(* Logix 5000 project; controller IndiconLLC vendor 1 type 14 code 77 rev 20.14; software revision 20.05 *)
// Indicon Emulation Department CompactLogix
// Development Kit PLC

TASK MainTask (continuous, watchdog 500 ms) : CPU

MODULES
   Controller : vendor 1 type 14 code 77 (CompactLogixL32EController 0, rev 20.14)
      LocalENB : 1769-L32E Ethernet Port (CompactLogixL32Ethernet 1, rev 20.11)
         AS1_ENBT : 1756-ENBT (Ethernet 192.168.112.83, rev 4.7, Output RPI 10 ms)
            AS1 : vendor 1 type 14 code 213 (ICP 2, rev 32.1, $37f21408$ RPI 50 ms)
      Local : CompactBus (CompactVirtualAdapter 3, rev 20.11)
END_MODULES

TYPE Emulation_Carrier_Object :
STRUCT
   Spawned : BOOL;
   XPos : DINT;
   Width : DINT;
   ZeroPoint : DINT;
   EndPoint : DINT;
   RealPosition : REAL;
   RestrictSpawn : BOOL;
   AttachedFront : BOOL;
   AttachedFrontID : DINT;
   AttachedRear : BOOL;
   AttachedRearID : DINT;
   DirectiveFlowFwd : BOOL;
   DirectiveFlowRev : BOOL;
   UpdateCounter : DINT;
END_STRUCT
END_TYPE

TYPE Emulation_Display_Env :
STRUCT
   Height : DINT;
   Width : DINT;
   CarrierObjectWidth : DINT;
   CarrierObjectCountSize : DINT;
   CarrierObjectFORControl : DINT;
   CarrierObjectFORControlEmbed : DINT;
   VFDObjectWidth : DINT;
   VFDObjectCountSize : DINT;
   VFDObjectFORControl : DINT;
END_STRUCT
END_TYPE

TYPE ProdCons_VFD :
STRUCT
   VFD : ProdCons_VFD_PTP_Setup[3];
END_STRUCT
END_TYPE

TYPE ProdCons_VFD_PTP_Setup :
STRUCT
   In : z_VFD_PTP_Emulation_Input;
   Out : z_VFD_PTP_Emulation_Output;
END_STRUCT
END_TYPE

TYPE ProdCons_VFD_Setup :
STRUCT
   In : z_VFD_Emulation_Input;
   Out : z_VFD_Emulation_Output;
END_STRUCT
END_TYPE

TYPE student_DataHandlingVehicleObject :
STRUCT
   Visibility : BOOL;
   YPosition : DINT;
   XPosition : DINT;
   PositionUpdateDwell : TIMER;
   InSpawnZone : BOOL;
   ShiftRegisterData : DINT;
   Color : SINT;
   ONS : DINT;
   DedicatedBank : SINT;
END_STRUCT
END_TYPE

TYPE z_VFD_Emulation :
STRUCT
   OverView : z_VFD_Emulation_Handling;
   MotorOutputs : z_VFD_Emulation_Input;
   MotorInputs : z_VFD_Emulation_Output;
END_STRUCT
END_TYPE

TYPE z_VFD_Emulation_Handling :
STRUCT
   XPosition : DINT;
   YPosition : DINT;
   Width : DINT;
   ZeroPoint : DINT;
   EndPoint : DINT;
   MoveFwd : BOOL;
   MoveRev : BOOL;
   HiSpeed : DINT;
   LoSpeed : DINT;
   HiSpeedEnable : BOOL;
   AccelRamp : DINT;
   DecelRamp : DINT;
   AccelCalc : REAL;
   DecelCalc : REAL;
   CurrentSpeed : REAL;
   SpeedCalc : REAL;
   ForwardLocked : BOOL;
   ReverseLocked : BOOL;
   PositionUpdateDwell : TIMER;
   SpeedDividend : REAL;
   IO : SINT;
   StationType : DINT;
   PXS : z_VFD_Emulation_IO_Handling[6];
   Position : DINT;
END_STRUCT
END_TYPE

TYPE z_VFD_Emulation_Input :
STRUCT
   ReadyToRun : BOOL;
   FaultCode : DINT;
   VelocityFeedback : DINT;
   MotorRunningFwd : BOOL;
   MotorRunningRev : BOOL;
   IO : SINT;
   PositionFeedback : DINT;
END_STRUCT
END_TYPE

TYPE z_VFD_Emulation_IO_Handling :
STRUCT
   Enable : BOOL;
   Position : DINT;
   RequestStuckOnSim : BOOL;
   RequestStuckOffSim : BOOL;
END_STRUCT
END_TYPE

TYPE z_VFD_Emulation_Output :
STRUCT
   RunForward : BOOL;
   RunReverse : BOOL;
   SpeedSetpoint : DINT;
   FaultReset : BOOL;
END_STRUCT
END_TYPE

TYPE z_VFD_PTP_Emulation :
STRUCT
   OverView : z_VFD_Emulation_Handling;
   MotorOutputs : z_VFD_PTP_Emulation_Input;
   MotorInputs : z_VFD_PTP_Emulation_Output;
END_STRUCT
END_TYPE

TYPE z_VFD_PTP_Emulation_Input :
STRUCT
   ReadyToRun : BOOL;
   FaultCode : DINT;
   VelocityFeedback : DINT;
   MotorRunningFwd : BOOL;
   MotorRunningRev : BOOL;
   IO : SINT;
   PositionFeedback : DINT;
END_STRUCT
END_TYPE

TYPE z_VFD_PTP_Emulation_Internal :
STRUCT
   Offset : DINT;
   Position : DINT;
   CaptureOneShot : BOOL;
   ForwardMoveRequired : BOOL;
   ReverseMoveRequired : BOOL;
   HighSpeedEnable : BOOL;
   CreepSpeedEnable : BOOL;
   SpeedLimit : REAL;
   AbsTenPercent : REAL;
   AbsTenPercentNeg : REAL;
   AbsTenPercentEmb : REAL;
   AbsTenPercentEmbNeg : REAL;
   OneShot : DINT;
END_STRUCT
END_TYPE

TYPE z_VFD_PTP_Emulation_Output :
STRUCT
   JogForward : BOOL;
   JogReverse : BOOL;
   SpeedSetpoint : DINT;
   PTPSetpoint : DINT;
   PTP_Move : BOOL;
   Run : BOOL;
   FaultReset : BOOL;
END_STRUCT
END_TYPE

TYPE zFlash :
STRUCT
   Slow : BOOL;
   Norm : BOOL;
   Fast : BOOL;
   Timer : TIMER;
END_STRUCT
END_TYPE

TYPE zTime :
STRUCT
   Year : DINT;
   Month : DINT;
   Day : DINT;
   Hour : DINT;
   Minute : DINT;
   Second : DINT;
   MSecond : DINT;
END_STRUCT
END_TYPE

VAR_GLOBAL   (* controller tags *)
   AS1_ToSupervisor : ProdCons_VFD := (VFD[0].Out.SpeedSetpoint := 500, VFD[0].Out.PTPSetpoint := 7718, VFD[1].Out.SpeedSetpoint := 250, VFD[1].Out.PTPSetpoint := 6082, VFD[2].Out.SpeedSetpoint := 250);
   Flash : zFlash := (Slow := 1, Fast := 1, Timer.PRE := 8388608, Timer.ACC := 3363, Timer.EN := 1, Timer.TT := 1);
   initializeDint : DINT := 100;
   InitializeMessage : MESSAGE;
        MessageParameters(ServiceCode := 16#004d, LocalElement := initializeDint, ...)
   ProducedData : DINT[300] := ([0] := 17);
   ReadWallClock : zTime := (Year := 2019, Month := 5, Day := 15, Hour := 4, Minute := 41, Second := 27, MSecond := 192466);
   Supervisor_ToAS1 : ProdCons_VFD := (VFD[0].In.PositionFeedback := 7718, VFD[1].In.PositionFeedback := 6082, VFD[2].In.PositionFeedback := 4); {produced}
   TempDINT : DINT[1000] := ([0] := 99999999, [1] := 99999999, [2] := 99999999, [3] := 99999999, [4] := 99999999, [5] := 99999999, [6] := 99999999, [7] := 99999999, [8] := 99999999, [9] := 99999999, [10] := 99999999, [11] := 99999999, [12] := 99999999, [13] := 99999999, [14] := 99999999, [15] := 99999999, [16] := 99999999, [17] := 99999999, [18] := 99999999, [19] := 99999999, [20] := 99999999, [21] := 99999999, [22] := 99999999, [23] := 99999999, [24] := 99999999, [25] := 99999999, [26] := 99999999, [27] := 99999999, [28] := 99999999, [29] := 99999999, [30] := 99999999, [31] := 99999999, [32] := 99999999, [33] := 99999999, [34] := 99999999, [35] := 99999999, [36] := 99999999, [37] := 99999999, [38] := 99999999, [39] := 99999999, [40] := 99999999, [41] := 99999999, [42] := 99999999, [43] := 99999999, [44] := 99999999, [45] := 99999999, [46] := 99999999, [47] := 99999999, [48] := 99999999, [49] := 99999999, [50] := 99999999, [51] := 99999999, [52] := 99999999, [53] := 99999999, [54] := 99999999, [55] := 99999999, [56] := 99999999, [57] := 99999999, [58] := 99999999, [59] := 99999999,
        [60] := 99999999, [61] := 99999999, [62] := 99999999, [63] := 99999999, [64] := 99999999, [65] := 99999999, [66] := 99999999, [67] := 99999999, [68] := 99999999, [69] := 99999999, [70] := 99999999, [71] := 99999999, [72] := 99999999, [73] := 99999999, [74] := 99999999, [75] := 99999999, [76] := 99999999, [77] := 99999999, [78] := 99999999, [79] := 99999999, [80] := 99999999, [81] := 99999999, [82] := 99999999, [83] := 99999999, [84] := 99999999, [85] := 99999999, [86] := 99999999, [87] := 99999999, [88] := 99999999, [89] := 99999999, [90] := 99999999, [91] := 99999999, [92] := 99999999, [93] := 99999999, [94] := 99999999, [95] := 99999999, [96] := 99999999, [97] := 99999999, [98] := 99999999, [99] := 99999999, [100] := 99999999, [101] := 99999999, [102] := 99999999, [103] := 99999999, [104] := 99999999, [105] := 99999999, [106] := 99999999, [107] := 99999999, [108] := 99999999, [109] := 99999999, [110] := 99999999, [111] := 99999999, [112] := 99999999, [113] := 99999999, [114] := 99999999, [115] := 99999999, [116] := 99999999, [117] := 99999999, [118] := 99999999, [119] := 99999999,
        [120] := 99999999, [121] := 99999999, [122] := 99999999, [123] := 99999999, [124] := 99999999, [125] := 99999999, [126] := 99999999, [127] := 99999999);
   TempINT : INT[1000] := ([0] := -7937, [1] := 1525, [2] := -7937, [3] := 1525, [4] := -7937, [5] := 1525, [6] := -7937, [7] := 1525, [8] := -7937, [9] := 1525, [10] := -7937, [11] := 1525, [12] := -7937, [13] := 1525, [14] := -7937, [15] := 1525, [16] := -7937, [17] := 1525, [18] := -7937, [19] := 1525, [20] := -7937, [21] := 1525, [22] := -7937, [23] := 1525, [24] := -7937, [25] := 1525, [26] := -7937, [27] := 1525, [28] := -7937, [29] := 1525, [30] := -7937, [31] := 1525, [32] := -7937, [33] := 1525, [34] := -7937, [35] := 1525, [36] := -7937, [37] := 1525, [38] := -7937, [39] := 1525, [40] := -7937, [41] := 1525, [42] := -7937, [43] := 1525, [44] := -7937, [45] := 1525, [46] := -7937, [47] := 1525, [48] := -7937, [49] := 1525, [50] := -7937, [51] := 1525, [52] := -7937, [53] := 1525, [54] := -7937, [55] := 1525, [56] := -7937, [57] := 1525, [58] := -7937, [59] := 1525,
        [60] := -7937, [61] := 1525, [62] := -7937, [63] := 1525, [64] := -7937, [65] := 1525, [66] := -7937, [67] := 1525, [68] := -7937, [69] := 1525, [70] := -7937, [71] := 1525, [72] := -7937, [73] := 1525, [74] := -7937, [75] := 1525, [76] := -7937, [77] := 1525, [78] := -7937, [79] := 1525, [80] := -7937, [81] := 1525, [82] := -7937, [83] := 1525, [84] := -7937, [85] := 1525, [86] := -7937, [87] := 1525, [88] := -7937, [89] := 1525, [90] := -7937, [91] := 1525, [92] := -7937, [93] := 1525, [94] := -7937, [95] := 1525, [96] := -7937, [97] := 1525, [98] := -7937, [99] := 1525, [100] := -7937, [101] := 1525, [102] := -7937, [103] := 1525, [104] := -7937, [105] := 1525, [106] := -7937, [107] := 1525, [108] := -7937, [109] := 1525, [110] := -7937, [111] := 1525, [112] := -7937, [113] := 1525, [114] := -7937, [115] := 1525, [116] := -7937, [117] := 1525, [118] := -7937, [119] := 1525,
        [120] := -7937, [121] := 1525, [122] := -7937, [123] := 1525, [124] := -7937, [125] := 1525, [126] := -7937, [127] := 1525);
   TempINT2 : INT[1000] := ([0] := -7937, [1] := 1525, [2] := -7937, [3] := 1525, [4] := -7937, [5] := 1525, [6] := -7937, [7] := 1525, [8] := -7937, [9] := 1525, [10] := -7937, [11] := 1525, [12] := -7937, [13] := 1525, [14] := -7937, [15] := 1525, [16] := -7937, [17] := 1525, [18] := -7937, [19] := 1525, [20] := -7937, [21] := 1525, [22] := -7937, [23] := 1525, [24] := -7937, [25] := 1525, [26] := -7937, [27] := 1525, [28] := -7937, [29] := 1525, [30] := -7937, [31] := 1525, [32] := -7937, [33] := 1525, [34] := -7937, [35] := 1525, [36] := -7937, [37] := 1525, [38] := -7937, [39] := 1525, [40] := -7937, [41] := 1525, [42] := -7937, [43] := 1525, [44] := -7937, [45] := 1525, [46] := -7937, [47] := 1525, [48] := -7937, [49] := 1525, [50] := -7937, [51] := 1525, [52] := -7937, [53] := 1525, [54] := -7937, [55] := 1525, [56] := -7937, [57] := 1525, [58] := -7937, [59] := 1525,
        [60] := -7937, [61] := 1525, [62] := -7937, [63] := 1525, [64] := -7937, [65] := 1525, [66] := -7937, [67] := 1525, [68] := -7937, [69] := 1525, [70] := -7937, [71] := 1525, [72] := -7937, [73] := 1525, [74] := -7937, [75] := 1525, [76] := -7937, [77] := 1525, [78] := -7937, [79] := 1525, [80] := -7937, [81] := 1525, [82] := -7937, [83] := 1525, [84] := -7937, [85] := 1525, [86] := -7937, [87] := 1525, [88] := -7937, [89] := 1525, [90] := -7937, [91] := 1525, [92] := -7937, [93] := 1525, [94] := -7937, [95] := 1525, [96] := -7937, [97] := 1525, [98] := -7937, [99] := 1525, [100] := -7937, [101] := 1525, [102] := -7937, [103] := 1525, [104] := -7937, [105] := 1525, [106] := -7937, [107] := 1525, [108] := -7937, [109] := 1525, [110] := -7937, [111] := 1525, [112] := -7937, [113] := 1525, [114] := -7937, [115] := 1525, [116] := -7937, [117] := 1525, [118] := -7937, [119] := 1525,
        [120] := -7937, [121] := 1525, [122] := -7937, [123] := 1525, [124] := -7937, [125] := 1525, [126] := -7937, [127] := 1525);
   VFDObject : z_VFD_PTP_Emulation[3] := ([0].OverView.AccelRamp := 10, [0].OverView.DecelRamp := 10, [0].OverView.AccelCalc := 0.1, [0].OverView.DecelCalc := 0.1, [0].OverView.SpeedCalc := 10.0, [0].OverView.PositionUpdateDwell.PRE := 10, [0].OverView.PositionUpdateDwell.ACC := 1, [0].OverView.PositionUpdateDwell.EN := 1, [0].OverView.PositionUpdateDwell.TT := 1, [0].MotorOutputs.PositionFeedback := 7718, [0].MotorInputs.SpeedSetpoint := 500, [0].MotorInputs.PTPSetpoint := 7718, [1].OverView.AccelRamp := 10, [1].OverView.DecelRamp := 10, [1].OverView.AccelCalc := 0.1, [1].OverView.DecelCalc := 0.1, [1].OverView.SpeedCalc := 10.0, [1].OverView.PositionUpdateDwell.PRE := 10, [1].OverView.PositionUpdateDwell.ACC := 2, [1].OverView.PositionUpdateDwell.EN := 1, [1].OverView.PositionUpdateDwell.TT := 1, [1].MotorOutputs.PositionFeedback := 6082, [1].MotorInputs.SpeedSetpoint := 250, [1].MotorInputs.PTPSetpoint := 6082, [2].OverView.AccelRamp := 10, [2].OverView.DecelRamp := 10, [2].OverView.AccelCalc := 0.1, [2].OverView.DecelCalc := 0.1, [2].OverView.SpeedCalc := 10.0, [2].OverView.PositionUpdateDwell.PRE := 10, [2].OverView.PositionUpdateDwell.ACC := 3, [2].OverView.PositionUpdateDwell.EN := 1, [2].OverView.PositionUpdateDwell.TT := 1, [2].MotorOutputs.PositionFeedback := 4, [2].MotorInputs.SpeedSetpoint := 250);
   VFDObjectInternal : z_VFD_PTP_Emulation_Internal[3] := ([0].Position := 7718, [0].CreepSpeedEnable := 1, [0].SpeedLimit := 10.0, [0].AbsTenPercentEmbNeg := -122.83199, [1].Position := 6082, [1].CreepSpeedEnable := 1, [1].SpeedLimit := 10.0, [1].AbsTenPercent := 74.5, [1].AbsTenPercentEmb := 18.625, [1].AbsTenPercentEmbNeg := 65.712, [2].Position := 4, [2].CreepSpeedEnable := 1, [2].SpeedLimit := 10.0);
   WallClock : zTime := (Year := 2002, Month := 12, Day := 3, Hour := 2, Minute := 11, Second := 30, MSecond := 968666);
   zz_irox : BOOL;
   zz_irox_dint : DINT := 3;
END_VAR

PROGRAM CPU   (* main routine A000_MainRoutine *)

ROUTINE A000_MainRoutine   (* ladder *)
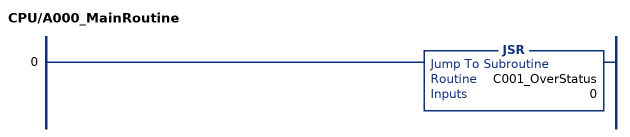
   0: JSR(C001_OverStatus,0);
END_ROUTINE

ROUTINE C001_OverStatus   (* ladder *)
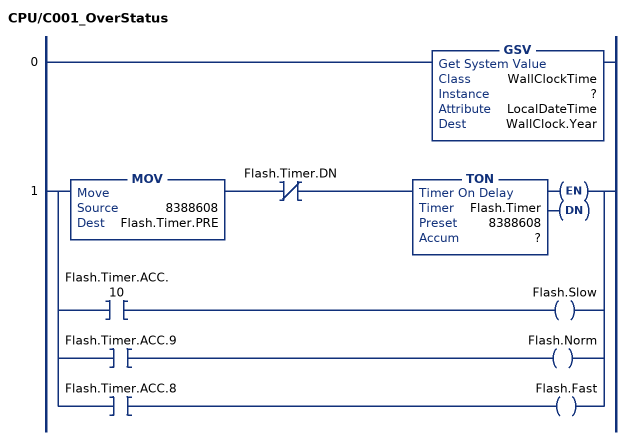
   0: GSV(WallClockTime,?,LocalDateTime,WallClock.Year);
   1: [MOV(8388608,Flash.Timer.PRE) XIO(Flash.Timer.DN) TON(Flash.Timer,?,?) ,XIC(Flash.Timer.ACC.10) OTE(Flash.Slow) ,XIC(Flash.Timer.ACC.9) OTE(Flash.Norm) ,XIC(Flash.Timer.ACC.8) OTE(Flash.Fast) ];
END_ROUTINE
END_PROGRAM

PROGRAM Testing_Environment   (* main routine MainRoutine *)
VAR
   AbsolueMoveDiagram : DINT := 899;
   AbsolueMoveDiagramReal : REAL;
   AbsoluteTenPercent : REAL;
   AbsoluteTenPercentSecondary : REAL;
   AccelDint : DINT := 10;
   Accelerate : BOOL;
   BargeEnable : BOOL;
   CarrierObjectLocal : Emulation_Carrier_Object := (XPos := 93, Width := 100, ZeroPoint := 93, EndPoint := 193, RealPosition := 92.9388, DirectiveFlowFwd := 1, DirectiveFlowRev := 1);
   ClockedDiagram : DINT := 89;
   CompareDint : DINT;
   CurrentClockedDiag : DINT;
   CurrentClockStep : DINT := 999;
   DataCalcd : BOOL := 1;
   Decelerate : BOOL;
   DeSpawnZone : DINT := 830;
   DisplayEnv : Emulation_Display_Env := (Height := 768, Width := 1200, CarrierObjectWidth := 100, CarrierObjectCountSize := 10, CarrierObjectFORControl := 3, VFDObjectCountSize := 12, VFDObjectFORControl := 12);
   DistanceTraveled : DINT;
   HiSpeedTestEnable : BOOL := 1;
   HoldSpeed : BOOL;
   InitializeEnvironment : BOOL;
   InitializeEnvironmentOneShot : DINT := 1;
   LocalMotor : z_VFD_Emulation := (OverView.AccelRamp := 1000, OverView.DecelRamp := 200, OverView.AccelCalc := 10.0, OverView.DecelCalc := 2.0, OverView.PositionUpdateDwell.PRE := 10, OverView.PositionUpdateDwell.ACC := 9, OverView.PositionUpdateDwell.EN := 1, OverView.PositionUpdateDwell.TT := 1, OverView.PXS[1].Position := 92, OverView.PXS[2].Position := 102, OverView.PXS[3].Position := 115, OverView.PXS[4].Position := 10, OverView.PXS[5].Position := -10, MotorOutputs.ReadyToRun := 1);
   LocalObject : Emulation_Carrier_Object := (Width := 100, EndPoint := 100, RestrictSpawn := 1);
   LocalPTPInternal : z_VFD_PTP_Emulation_Internal := (Position := 4, CreepSpeedEnable := 1, SpeedLimit := 10.0);
   LocalPTPMotor : z_VFD_PTP_Emulation := (OverView.AccelRamp := 10, OverView.DecelRamp := 10, OverView.AccelCalc := 0.1, OverView.DecelCalc := 0.1, OverView.SpeedCalc := 10.0, OverView.PositionUpdateDwell.PRE := 10, OverView.PositionUpdateDwell.ACC := 3, OverView.PositionUpdateDwell.EN := 1, OverView.PositionUpdateDwell.TT := 1, MotorOutputs.PositionFeedback := 4, MotorInputs.SpeedSetpoint := 250);
   LongEnable : BOOL;
   LoSpeedTestEnable : BOOL;
   MoveComplete : BOOL := 1;
   PassThroughStationEnable : BOOL;
   PositionClock : DINT := 89;
   ReqAccelStamp : DINT := 18;
   ReqAccelStampReal : REAL;
   ReqDecelStamp : DINT := 18;
   ReqDecelStampReal : REAL;
   ReqDecelStartClock : DINT := 71;
   TestBit : BOOL;
   TestBit2 : BOOL := 1;
   VFD_PTP_Internal : z_VFD_PTP_Emulation_Internal := (CaptureOneShot := 1);
   VFD_PTPObject : z_VFD_PTP_Emulation := (OverView.AccelRamp := 1000, OverView.DecelRamp := 1000, OverView.AccelCalc := 10.0, OverView.DecelCalc := 10.0, OverView.PositionUpdateDwell.PRE := 10, OverView.PositionUpdateDwell.EN := 1, OverView.PositionUpdateDwell.TT := 1);
   VFDObjectWidth : DINT := 122;
END_VAR

ROUTINE B001_BufferIn   (* ladder *)
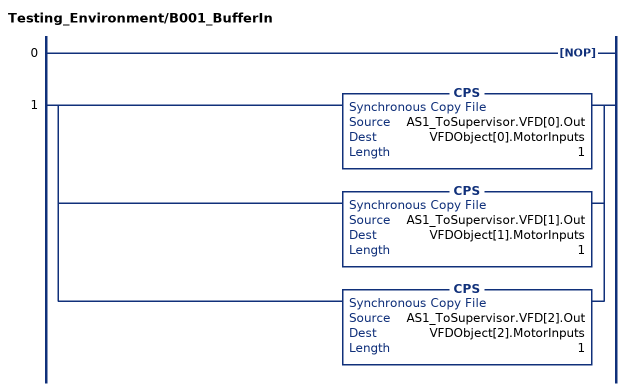
   0: NOP();
   1: [CPS(AS1_ToSupervisor.VFD[0].Out,VFDObject[0].MotorInputs,1) ,CPS(AS1_ToSupervisor.VFD[1].Out,VFDObject[1].MotorInputs,1) ,CPS(AS1_ToSupervisor.VFD[2].Out,VFDObject[2].MotorInputs,1) ];
END_ROUTINE

ROUTINE B002_BufferOut   (* ladder *)
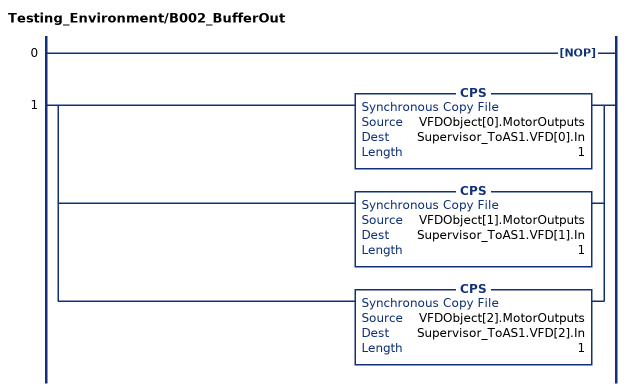
   0: NOP();
   1: [CPS(VFDObject[0].MotorOutputs,Supervisor_ToAS1.VFD[0].In,1) ,CPS(VFDObject[1].MotorOutputs,Supervisor_ToAS1.VFD[1].In,1) ,CPS(VFDObject[2].MotorOutputs,Supervisor_ToAS1.VFD[2].In,1) ];
END_ROUTINE

ROUTINE DTAP_Test   (* ladder *)
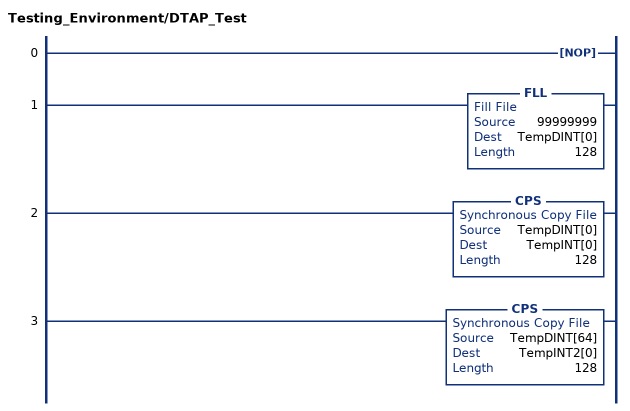
   0: NOP();
   1: FLL(99999999,TempDINT[0],128);
   2: CPS(TempDINT[0],TempINT[0],128);
   3: CPS(TempDINT[64],TempINT2[0],128);
END_ROUTINE

ROUTINE M001_Drive_Motors   (* ladder *)
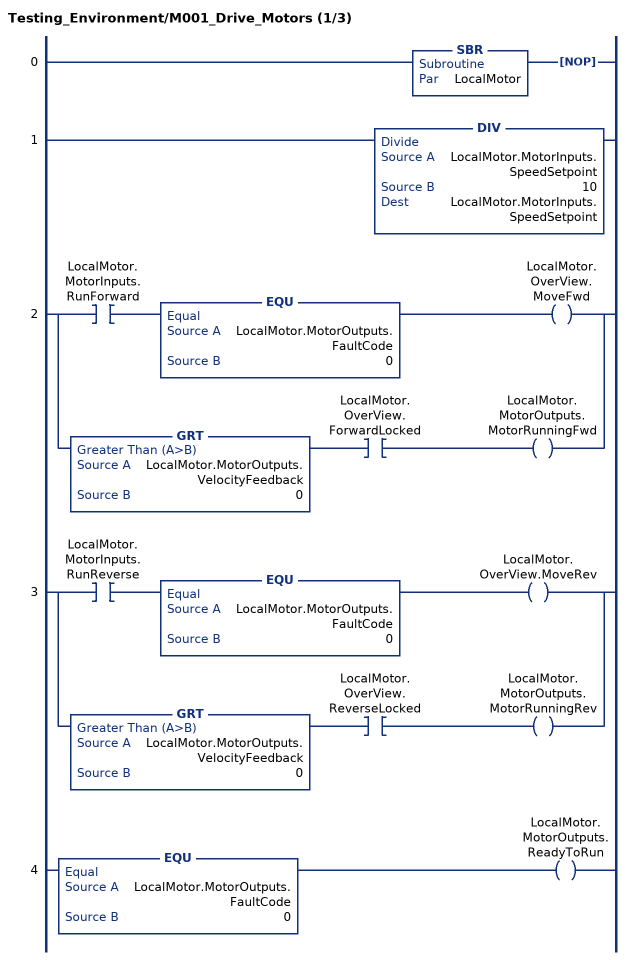
   0: SBR(LocalMotor)NOP();
   1: DIV(LocalMotor.MotorInputs.SpeedSetpoint,10,LocalMotor.MotorInputs.SpeedSetpoint);
   2: [XIC(LocalMotor.MotorInputs.RunForward) EQU(LocalMotor.MotorOutputs.FaultCode,0) OTE(LocalMotor.OverView.MoveFwd) ,GRT(LocalMotor.MotorOutputs.VelocityFeedback,0) XIC(LocalMotor.OverView.ForwardLocked) OTE(LocalMotor.MotorOutputs.MotorRunningFwd) ];
   3: [XIC(LocalMotor.MotorInputs.RunReverse) EQU(LocalMotor.MotorOutputs.FaultCode,0) OTE(LocalMotor.OverView.MoveRev) ,GRT(LocalMotor.MotorOutputs.VelocityFeedback,0) XIC(LocalMotor.OverView.ReverseLocked) OTE(LocalMotor.MotorOutputs.MotorRunningRev) ];
   4: EQU(LocalMotor.MotorOutputs.FaultCode,0)OTE(LocalMotor.MotorOutputs.ReadyToRun);
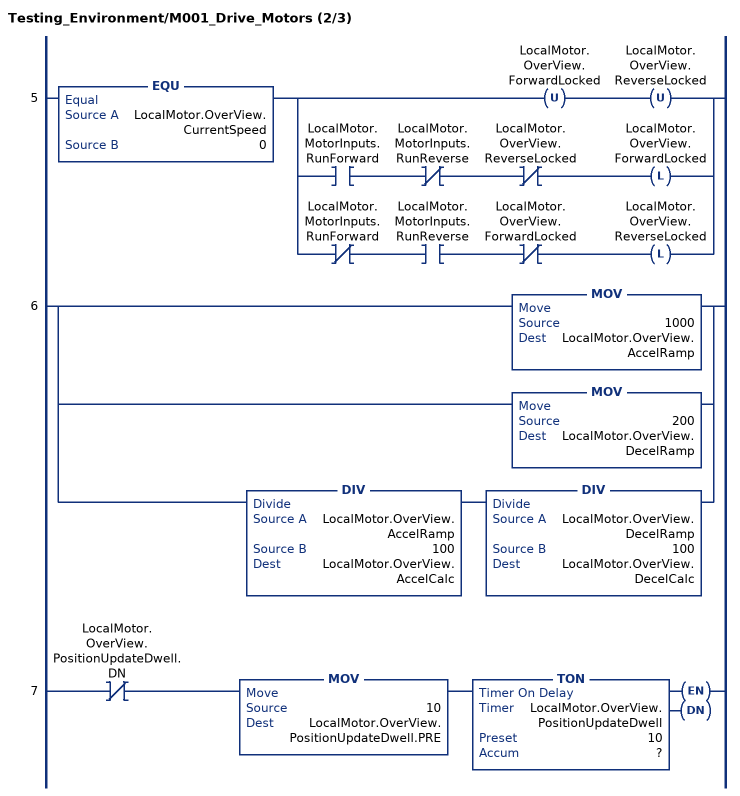
   5: EQU(LocalMotor.OverView.CurrentSpeed,0)[OTU(LocalMotor.OverView.ForwardLocked) OTU(LocalMotor.OverView.ReverseLocked) ,XIC(LocalMotor.MotorInputs.RunForward) XIO(LocalMotor.MotorInputs.RunReverse) XIO(LocalMotor.OverView.ReverseLocked) OTL(LocalMotor.OverView.ForwardLocked) ,XIO(LocalMotor.MotorInputs.RunForward) XIC(LocalMotor.MotorInputs.RunReverse) XIO(LocalMotor.OverView.ForwardLocked) OTL(LocalMotor.OverView.ReverseLocked) ];
   6: [MOV(1000,LocalMotor.OverView.AccelRamp) ,MOV(200,LocalMotor.OverView.DecelRamp) ,DIV(LocalMotor.OverView.AccelRamp,100,LocalMotor.OverView.AccelCalc) DIV(LocalMotor.OverView.DecelRamp,100,LocalMotor.OverView.DecelCalc) ];
   7: XIO(LocalMotor.OverView.PositionUpdateDwell.DN)MOV(10,LocalMotor.OverView.PositionUpdateDwell.PRE)TON(LocalMotor.OverView.PositionUpdateDwell,?,?);
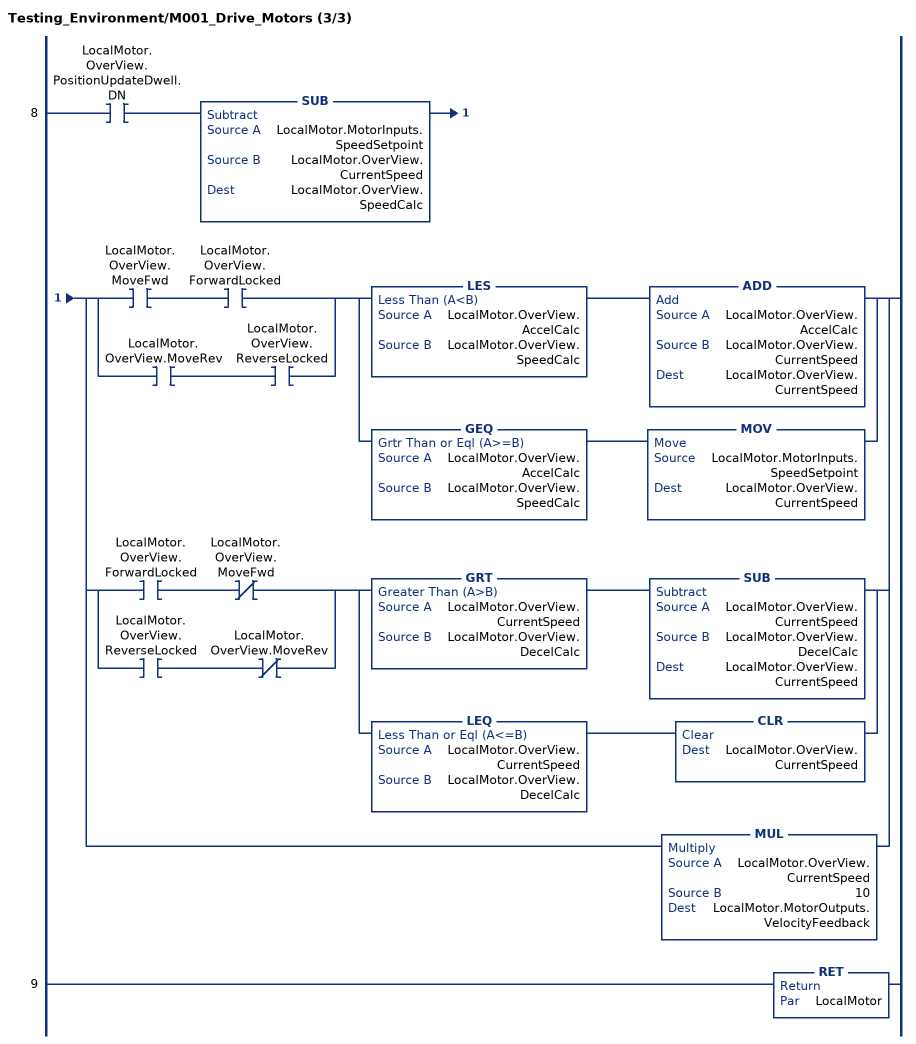
   8: XIC(LocalMotor.OverView.PositionUpdateDwell.DN)SUB(LocalMotor.MotorInputs.SpeedSetpoint,LocalMotor.OverView.CurrentSpeed,LocalMotor.OverView.SpeedCalc)[[XIC(LocalMotor.OverView.MoveFwd) XIC(LocalMotor.OverView.ForwardLocked) ,XIC(LocalMotor.OverView.MoveRev) XIC(LocalMotor.OverView.ReverseLocked) ] [LES(LocalMotor.OverView.AccelCalc,LocalMotor.OverView.SpeedCalc) ADD(LocalMotor.OverView.AccelCalc,LocalMotor.OverView.CurrentSpeed,LocalMotor.OverView.CurrentSpeed) ,GEQ(LocalMotor.OverView.AccelCalc,LocalMotor.OverView.SpeedCalc) MOV(LocalMotor.MotorInputs.SpeedSetpoint,LocalMotor.OverView.CurrentSpeed) ] ,[XIC(LocalMotor.OverView.ForwardLocked) XIO(LocalMotor.OverView.MoveFwd) ,XIC(LocalMotor.OverView.ReverseLocked) XIO(LocalMotor.OverView.MoveRev) ] [GRT(LocalMotor.OverView.CurrentSpeed,LocalMotor.OverView.DecelCalc) SUB(LocalMotor.OverView.CurrentSpeed,LocalMotor.OverView.DecelCalc,LocalMotor.OverView.CurrentSpeed) ,LEQ(LocalMotor.OverView.CurrentSpeed,LocalMotor.OverView.DecelCalc) CLR(LocalMotor.OverView.CurrentSpeed) ] ,MUL(LocalMotor.OverView.CurrentSpeed,10,LocalMotor.MotorOutputs.VelocityFeedback) ];
   9: RET(LocalMotor);
END_ROUTINE

ROUTINE M002_Drive_PTP_Motors   (* ladder *)
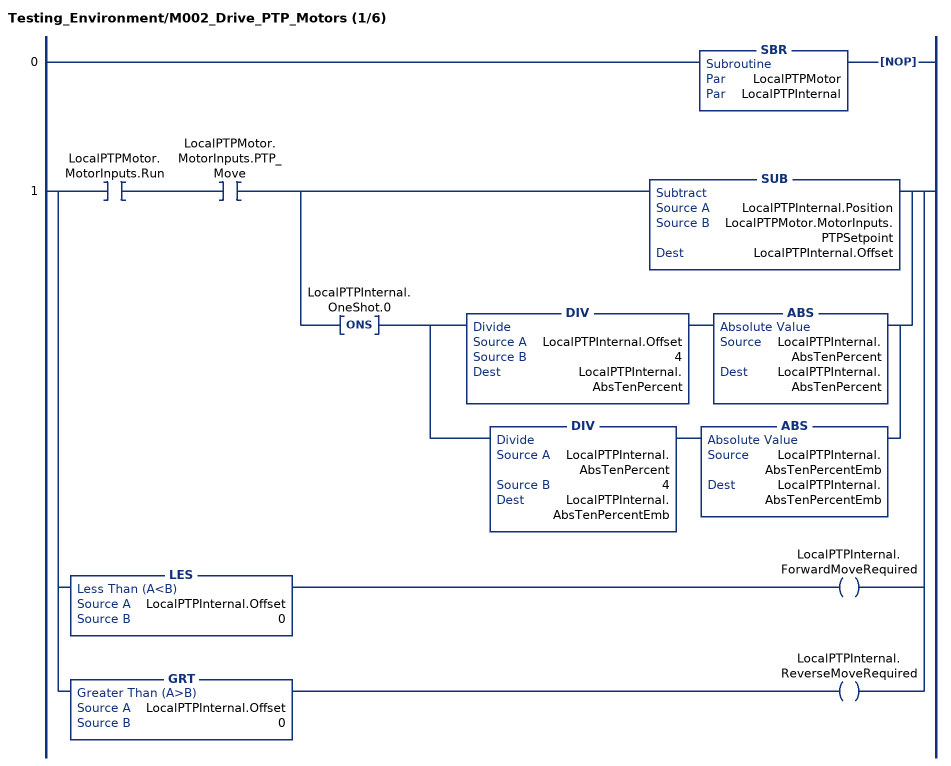
   0: SBR(LocalPTPMotor,LocalPTPInternal)NOP();
   1: [XIC(LocalPTPMotor.MotorInputs.Run) XIC(LocalPTPMotor.MotorInputs.PTP_Move) [SUB(LocalPTPInternal.Position,LocalPTPMotor.MotorInputs.PTPSetpoint,LocalPTPInternal.Offset) ,ONS(LocalPTPInternal.OneShot.0) [DIV(LocalPTPInternal.Offset,4,LocalPTPInternal.AbsTenPercent) ABS(LocalPTPInternal.AbsTenPercent,LocalPTPInternal.AbsTenPercent) ,DIV(LocalPTPInternal.AbsTenPercent,4,LocalPTPInternal.AbsTenPercentEmb) ABS(LocalPTPInternal.AbsTenPercentEmb,LocalPTPInternal.AbsTenPercentEmb) ] ] ,LES(LocalPTPInternal.Offset,0) OTE(LocalPTPInternal.ForwardMoveRequired) ,GRT(LocalPTPInternal.Offset,0) OTE(LocalPTPInternal.ReverseMoveRequired) ];
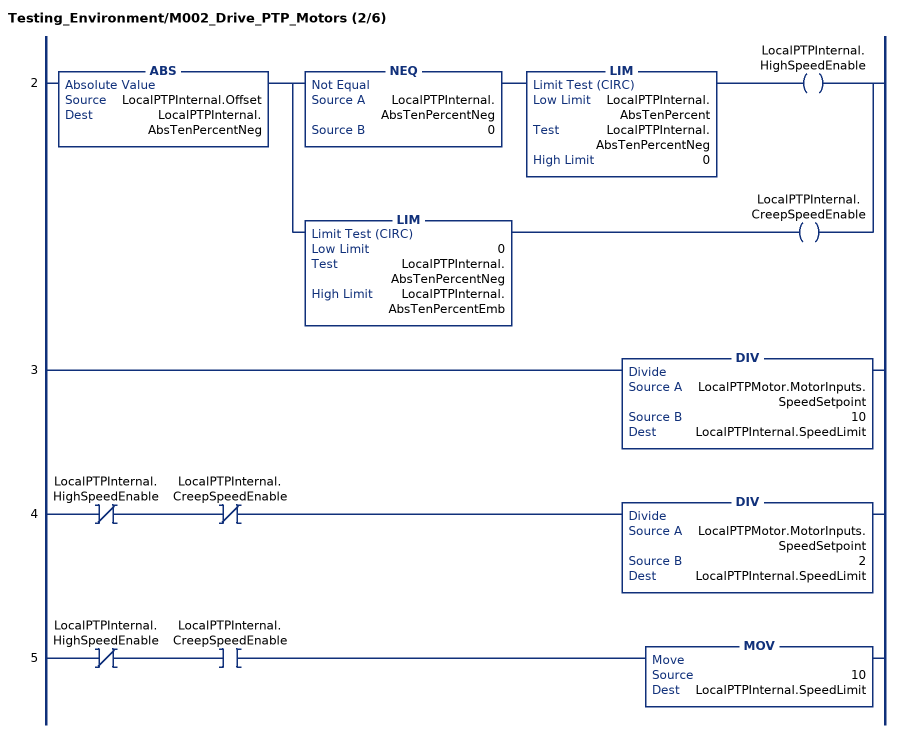
   2: ABS(LocalPTPInternal.Offset,LocalPTPInternal.AbsTenPercentNeg)[NEQ(LocalPTPInternal.AbsTenPercentNeg,0) LIM(LocalPTPInternal.AbsTenPercent,LocalPTPInternal.AbsTenPercentNeg,0) OTE(LocalPTPInternal.HighSpeedEnable) ,LIM(0,LocalPTPInternal.AbsTenPercentNeg,LocalPTPInternal.AbsTenPercentEmb) OTE(LocalPTPInternal.CreepSpeedEnable) ];
   3: DIV(LocalPTPMotor.MotorInputs.SpeedSetpoint,10,LocalPTPInternal.SpeedLimit);
   4: XIO(LocalPTPInternal.HighSpeedEnable)XIO(LocalPTPInternal.CreepSpeedEnable)DIV(LocalPTPMotor.MotorInputs.SpeedSetpoint,2,LocalPTPInternal.SpeedLimit);
   5: XIO(LocalPTPInternal.HighSpeedEnable)XIC(LocalPTPInternal.CreepSpeedEnable)MOV(10,LocalPTPInternal.SpeedLimit);
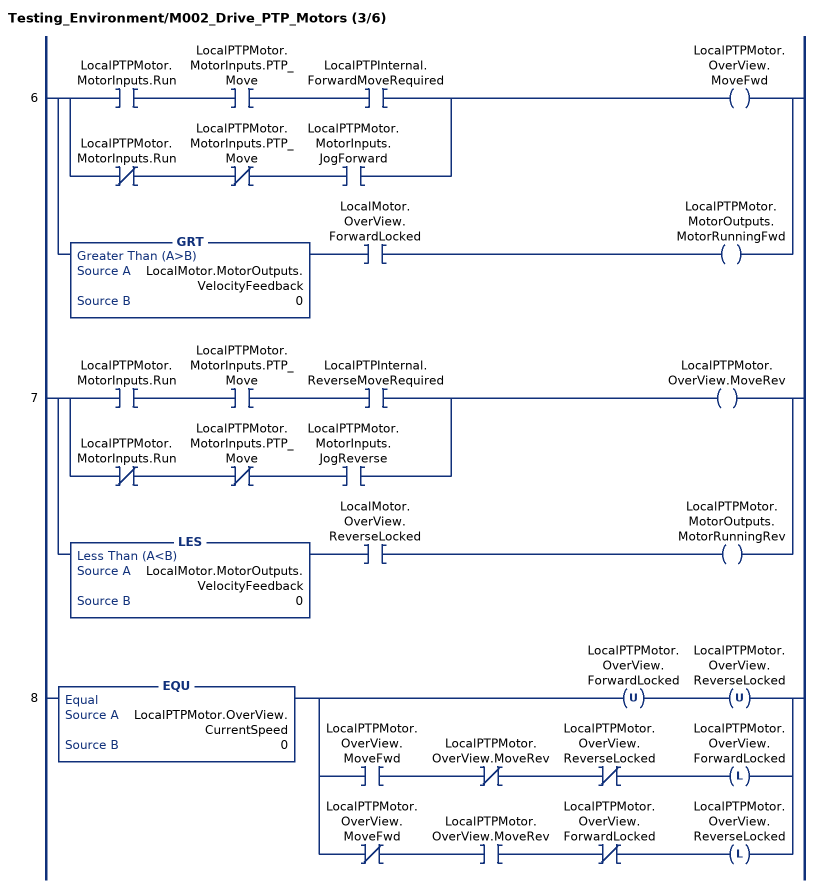
   6: [[XIC(LocalPTPMotor.MotorInputs.Run) XIC(LocalPTPMotor.MotorInputs.PTP_Move) XIC(LocalPTPInternal.ForwardMoveRequired) ,XIO(LocalPTPMotor.MotorInputs.Run) XIO(LocalPTPMotor.MotorInputs.PTP_Move) XIC(LocalPTPMotor.MotorInputs.JogForward) ] OTE(LocalPTPMotor.OverView.MoveFwd) ,GRT(LocalMotor.MotorOutputs.VelocityFeedback,0) XIC(LocalMotor.OverView.ForwardLocked) OTE(LocalPTPMotor.MotorOutputs.MotorRunningFwd) ];
   7: [[XIC(LocalPTPMotor.MotorInputs.Run) XIC(LocalPTPMotor.MotorInputs.PTP_Move) XIC(LocalPTPInternal.ReverseMoveRequired) ,XIO(LocalPTPMotor.MotorInputs.Run) XIO(LocalPTPMotor.MotorInputs.PTP_Move) XIC(LocalPTPMotor.MotorInputs.JogReverse) ] OTE(LocalPTPMotor.OverView.MoveRev) ,LES(LocalMotor.MotorOutputs.VelocityFeedback,0) XIC(LocalMotor.OverView.ReverseLocked) OTE(LocalPTPMotor.MotorOutputs.MotorRunningRev) ];
   8: EQU(LocalPTPMotor.OverView.CurrentSpeed,0)[OTU(LocalPTPMotor.OverView.ForwardLocked) OTU(LocalPTPMotor.OverView.ReverseLocked) ,XIC(LocalPTPMotor.OverView.MoveFwd) XIO(LocalPTPMotor.OverView.MoveRev) XIO(LocalPTPMotor.OverView.ReverseLocked) OTL(LocalPTPMotor.OverView.ForwardLocked) ,XIO(LocalPTPMotor.OverView.MoveFwd) XIC(LocalPTPMotor.OverView.MoveRev) XIO(LocalPTPMotor.OverView.ForwardLocked) OTL(LocalPTPMotor.OverView.ReverseLocked) ];
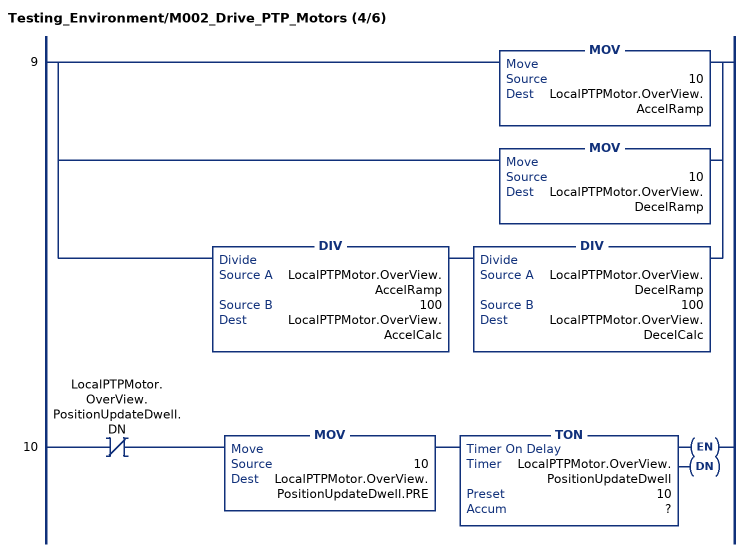
   9: [MOV(10,LocalPTPMotor.OverView.AccelRamp) ,MOV(10,LocalPTPMotor.OverView.DecelRamp) ,DIV(LocalPTPMotor.OverView.AccelRamp,100,LocalPTPMotor.OverView.AccelCalc) DIV(LocalPTPMotor.OverView.DecelRamp,100,LocalPTPMotor.OverView.DecelCalc) ];
   10: XIO(LocalPTPMotor.OverView.PositionUpdateDwell.DN)MOV(10,LocalPTPMotor.OverView.PositionUpdateDwell.PRE)TON(LocalPTPMotor.OverView.PositionUpdateDwell,?,?);
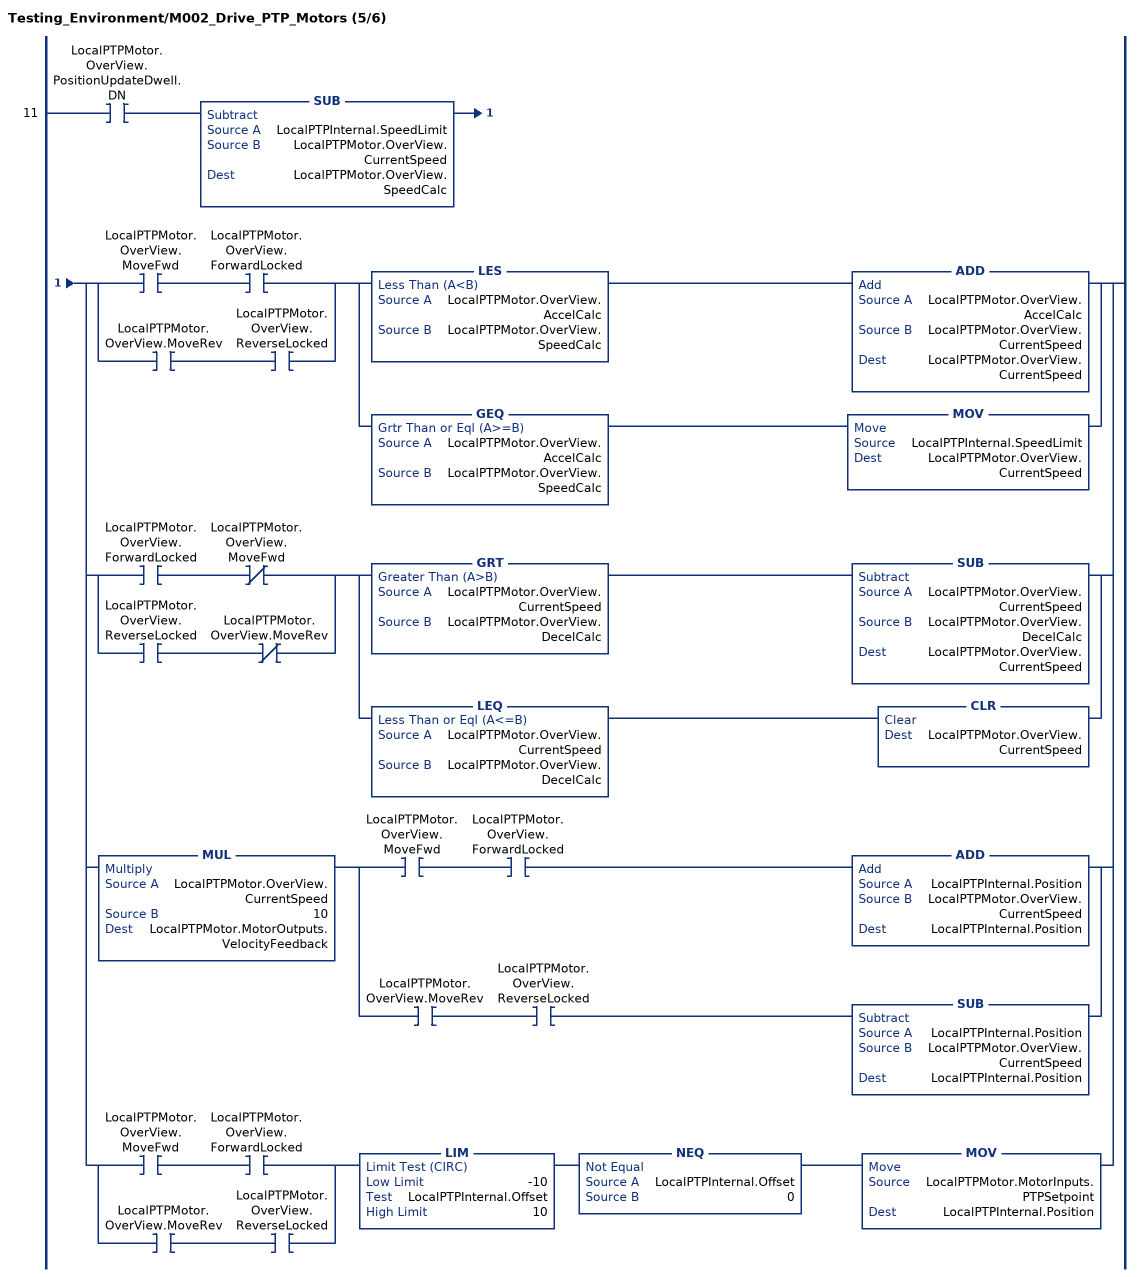
   11: XIC(LocalPTPMotor.OverView.PositionUpdateDwell.DN)SUB(LocalPTPInternal.SpeedLimit,LocalPTPMotor.OverView.CurrentSpeed,LocalPTPMotor.OverView.SpeedCalc)[[XIC(LocalPTPMotor.OverView.MoveFwd) XIC(LocalPTPMotor.OverView.ForwardLocked) ,XIC(LocalPTPMotor.OverView.MoveRev) XIC(LocalPTPMotor.OverView.ReverseLocked) ] [LES(LocalPTPMotor.OverView.AccelCalc,LocalPTPMotor.OverView.SpeedCalc) ADD(LocalPTPMotor.OverView.AccelCalc,LocalPTPMotor.OverView.CurrentSpeed,LocalPTPMotor.OverView.CurrentSpeed) ,GEQ(LocalPTPMotor.OverView.AccelCalc,LocalPTPMotor.OverView.SpeedCalc) MOV(LocalPTPInternal.SpeedLimit,LocalPTPMotor.OverView.CurrentSpeed) ] ,[XIC(LocalPTPMotor.OverView.ForwardLocked) XIO(LocalPTPMotor.OverView.MoveFwd) ,XIC(LocalPTPMotor.OverView.ReverseLocked) XIO(LocalPTPMotor.OverView.MoveRev) ] [GRT(LocalPTPMotor.OverView.CurrentSpeed,LocalPTPMotor.OverView.DecelCalc) SUB(LocalPTPMotor.OverView.CurrentSpeed,LocalPTPMotor.OverView.DecelCalc,LocalPTPMotor.OverView.CurrentSpeed) ,LEQ(LocalPTPMotor.OverView.CurrentSpeed,LocalPTPMotor.OverView.DecelCalc) CLR(LocalPTPMotor.OverView.CurrentSpeed) ] ,MUL(LocalPTPMotor.OverView.CurrentSpeed,10,LocalPTPMotor.MotorOutputs.VelocityFeedback) [XIC(LocalPTPMotor.OverView.MoveFwd) XIC(LocalPTPMotor.OverView.ForwardLocked) ADD(LocalPTPInternal.Position,LocalPTPMotor.OverView.CurrentSpeed,LocalPTPInternal.Position) ,XIC(LocalPTPMotor.OverView.MoveRev) XIC(LocalPTPMotor.OverView.ReverseLocked) SUB(LocalPTPInternal.Position,LocalPTPMotor.OverView.CurrentSpeed,LocalPTPInternal.Position) ] ,[XIC(LocalPTPMotor.OverView.MoveFwd) XIC(LocalPTPMotor.OverView.ForwardLocked) ,XIC(LocalPTPMotor.OverView.MoveRev) XIC(LocalPTPMotor.OverView.ReverseLocked) ] LIM(-10,LocalPTPInternal.Offset,10) NEQ(LocalPTPInternal.Offset,0) MOV(LocalPTPMotor.MotorInputs.PTPSetpoint,LocalPTPInternal.Position) ];
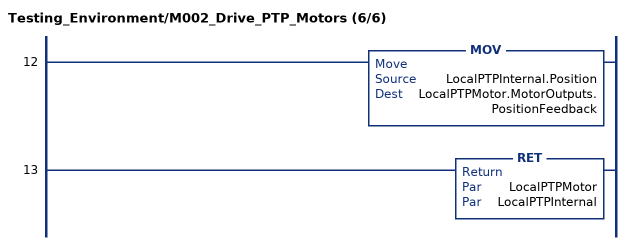
   12: MOV(LocalPTPInternal.Position,LocalPTPMotor.MotorOutputs.PositionFeedback);
   13: RET(LocalPTPMotor,LocalPTPInternal);
END_ROUTINE

ROUTINE MainRoutine   (* ladder *)
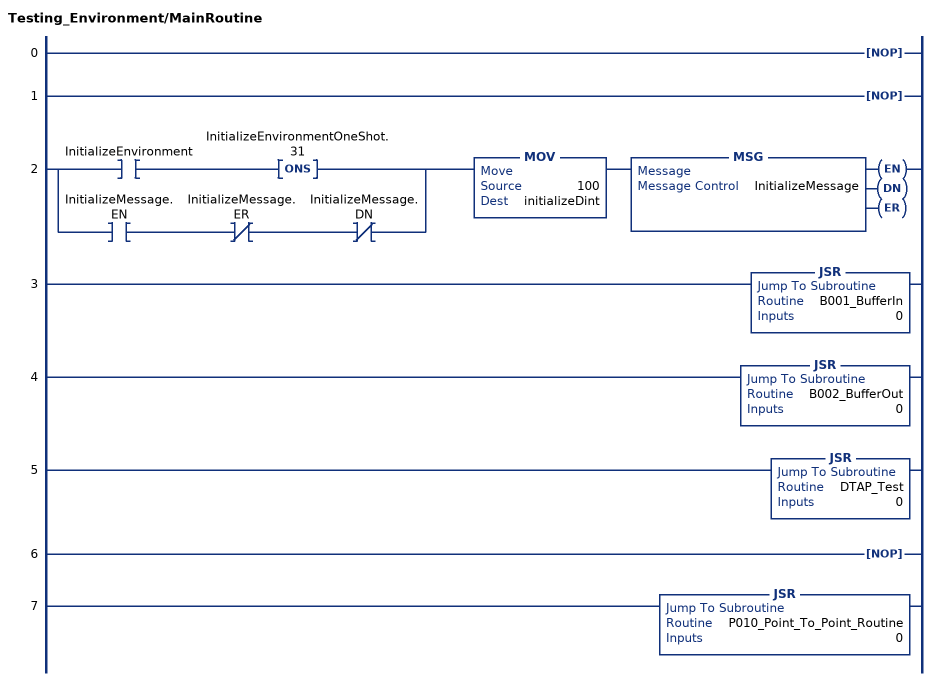
   0: NOP();
   1: NOP();
   2: [XIC(InitializeEnvironment) ONS(InitializeEnvironmentOneShot.31) ,XIC(InitializeMessage.EN) XIO(InitializeMessage.ER) XIO(InitializeMessage.DN) ]MOV(100,initializeDint)MSG(InitializeMessage);
   3: JSR(B001_BufferIn,0);
   4: JSR(B002_BufferOut,0);
   5: JSR(DTAP_Test,0);
   6: NOP();
   7: JSR(P010_Point_To_Point_Routine,0);
END_ROUTINE

ROUTINE N001_Carrier_Objects   (* ladder *)
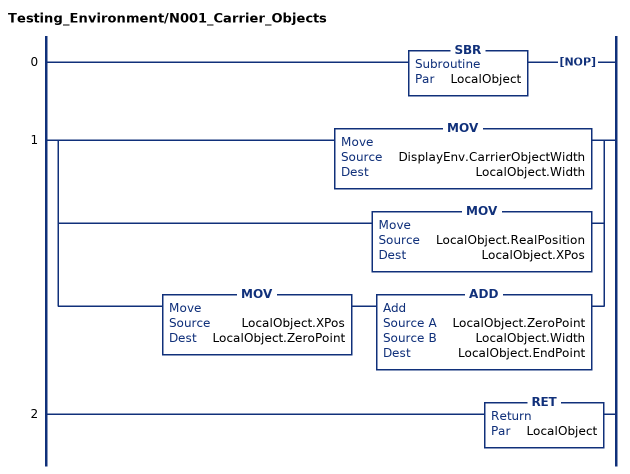
   0: SBR(LocalObject)NOP();
   1: [MOV(DisplayEnv.CarrierObjectWidth,LocalObject.Width) ,MOV(LocalObject.RealPosition,LocalObject.XPos) ,MOV(LocalObject.XPos,LocalObject.ZeroPoint) ADD(LocalObject.ZeroPoint,LocalObject.Width,LocalObject.EndPoint) ];
   2: RET(LocalObject);
END_ROUTINE

ROUTINE P010_Point_To_Point_Routine   (* ladder *)
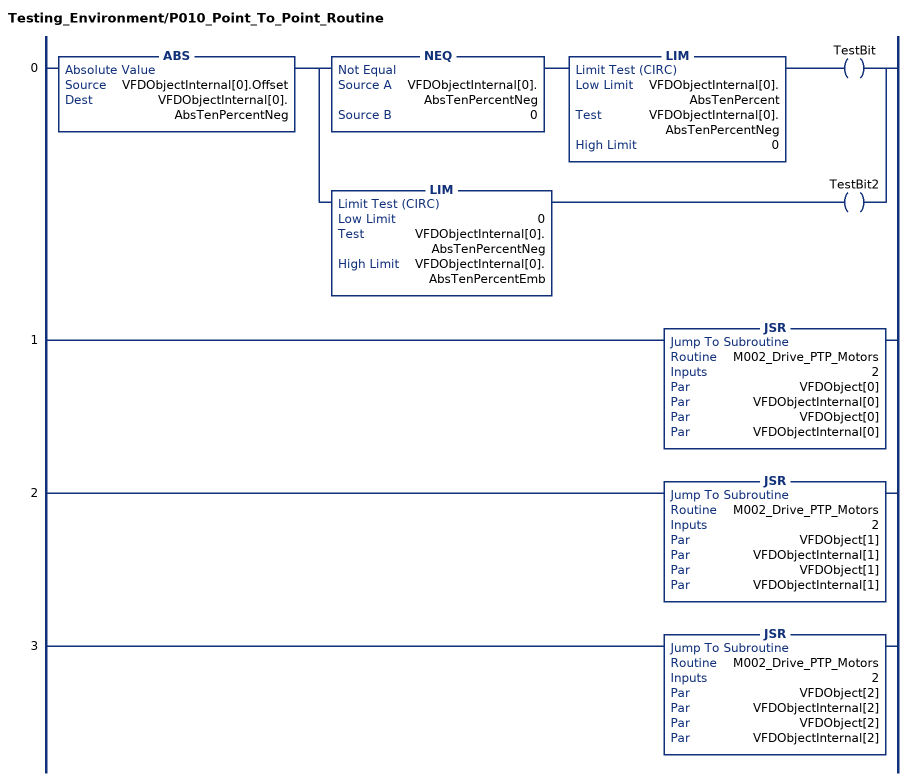
   0: ABS(VFDObjectInternal[0].Offset,VFDObjectInternal[0].AbsTenPercentNeg)[NEQ(VFDObjectInternal[0].AbsTenPercentNeg,0) LIM(VFDObjectInternal[0].AbsTenPercent,VFDObjectInternal[0].AbsTenPercentNeg,0) OTE(TestBit) ,LIM(0,VFDObjectInternal[0].AbsTenPercentNeg,VFDObjectInternal[0].AbsTenPercentEmb) OTE(TestBit2) ];
   1: JSR(M002_Drive_PTP_Motors,2,VFDObject[0],VFDObjectInternal[0],VFDObject[0],VFDObjectInternal[0]);
   2: JSR(M002_Drive_PTP_Motors,2,VFDObject[1],VFDObjectInternal[1],VFDObject[1],VFDObjectInternal[1]);
   3: JSR(M002_Drive_PTP_Motors,2,VFDObject[2],VFDObjectInternal[2],VFDObject[2],VFDObjectInternal[2]);
END_ROUTINE
END_PROGRAM
